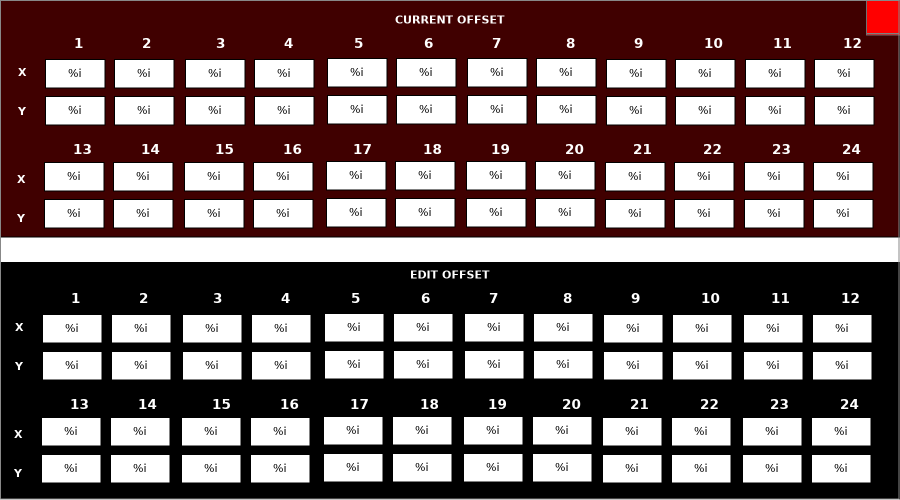
VISUALIZATION MOffset_1  // 900x500
    RoundedRectangle (0,0 900x237)
    Label (0,0 900x40), "CURRENT OFFSET"
    Label (15,55 25x35), "X"
    RoundedRectangle (45,59 60x29), "%i", text variable: Status_GVL.RecipeLine[1].OffsetPattern.Offset_X[1]
    Label (71,26 25x35), "1"
    RoundedRectangle (114,59 60x29), "%i", text variable: Status_GVL.RecipeLine[1].OffsetPattern.Offset_X[2]
    Label (139,26 25x35), "2"
    RoundedRectangle (185,59 60x29), "%i", text variable: Status_GVL.RecipeLine[1].OffsetPattern.Offset_X[3]
    RoundedRectangle (254,59 60x29), "%i", text variable: Status_GVL.RecipeLine[1].OffsetPattern.Offset_X[4]
    Label (15,94 25x35), "Y"
    RoundedRectangle (327,58 60x29), "%i", text variable: Status_GVL.RecipeLine[1].OffsetPattern.Offset_X[5]
    RoundedRectangle (396,58 60x29), "%i", text variable: Status_GVL.RecipeLine[1].OffsetPattern.Offset_X[6]
    RoundedRectangle (467,58 60x29), "%i", text variable: Status_GVL.RecipeLine[1].OffsetPattern.Offset_X[7]
    RoundedRectangle (536,58 60x29), "%i", text variable: Status_GVL.RecipeLine[1].OffsetPattern.Offset_X[8]
    RoundedRectangle (606,59 60x29), "%i", text variable: Status_GVL.RecipeLine[1].OffsetPattern.Offset_X[9]
    RoundedRectangle (675,59 60x29), "%i", text variable: Status_GVL.RecipeLine[1].OffsetPattern.Offset_X[10]
    Label (213,26 25x35), "3"
    Label (281,26 25x35), "4"
    Label (351,26 25x35), "5"
    Label (421,26 25x35), "6"
    Label (489,26 25x35), "7"
    Label (563,26 25x35), "8"
    Label (631,26 25x35), "9"
    Label (701,26 25x35), "10"
    RoundedRectangle (45,96 60x29), "%i", text variable: Status_GVL.RecipeLine[1].OffsetPattern.Offset_Y[1]
    RoundedRectangle (114,96 60x29), "%i", text variable: Status_GVL.RecipeLine[1].OffsetPattern.Offset_Y[2]
    RoundedRectangle (185,96 60x29), "%i", text variable: Status_GVL.RecipeLine[1].OffsetPattern.Offset_Y[3]
    RoundedRectangle (254,96 60x29), "%i", text variable: Status_GVL.RecipeLine[1].OffsetPattern.Offset_Y[4]
    RoundedRectangle (327,95 60x29), "%i", text variable: Status_GVL.RecipeLine[1].OffsetPattern.Offset_Y[5]
    RoundedRectangle (396,95 60x29), "%i", text variable: Status_GVL.RecipeLine[1].OffsetPattern.Offset_Y[6]
    RoundedRectangle (467,95 60x29), "%i", text variable: Status_GVL.RecipeLine[1].OffsetPattern.Offset_Y[7]
    RoundedRectangle (536,95 60x29), "%i", text variable: Status_GVL.RecipeLine[1].OffsetPattern.Offset_Y[8]
    RoundedRectangle (606,96 60x29), "%i", text variable: Status_GVL.RecipeLine[1].OffsetPattern.Offset_Y[9]
    RoundedRectangle (675,96 60x29), "%i", text variable: Status_GVL.RecipeLine[1].OffsetPattern.Offset_Y[10]
    Label (14,162 25x35), "X"
    RoundedRectangle (44,162 60x29), "%i", text variable: Status_GVL.RecipeLine[1].OffsetPattern.Offset_X[13]
    RoundedRectangle (113,162 60x29), "%i", text variable: Status_GVL.RecipeLine[1].OffsetPattern.Offset_X[14]
    RoundedRectangle (184,162 60x29), "%i", text variable: Status_GVL.RecipeLine[1].OffsetPattern.Offset_X[15]
    RoundedRectangle (253,162 60x29), "%i", text variable: Status_GVL.RecipeLine[1].OffsetPattern.Offset_X[16]
    Label (14,201 25x35), "Y"
    RoundedRectangle (326,161 60x29), "%i", text variable: Status_GVL.RecipeLine[1].OffsetPattern.Offset_X[17]
    RoundedRectangle (395,161 60x29), "%i", text variable: Status_GVL.RecipeLine[1].OffsetPattern.Offset_X[18]
    RoundedRectangle (466,161 60x29), "%i", text variable: Status_GVL.RecipeLine[1].OffsetPattern.Offset_X[19]
    RoundedRectangle (535,161 60x29), "%i", text variable: Status_GVL.RecipeLine[1].OffsetPattern.Offset_X[20]
    RoundedRectangle (605,162 60x29), "%i", text variable: Status_GVL.RecipeLine[1].OffsetPattern.Offset_X[21]
    RoundedRectangle (674,162 60x29), "%i", text variable: Status_GVL.RecipeLine[1].OffsetPattern.Offset_X[22]
    RoundedRectangle (44,199 60x29), "%i", text variable: Status_GVL.RecipeLine[1].OffsetPattern.Offset_Y[13]
    RoundedRectangle (113,199 60x29), "%i", text variable: Status_GVL.RecipeLine[1].OffsetPattern.Offset_Y[14]
    RoundedRectangle (184,199 60x29), "%i", text variable: Status_GVL.RecipeLine[1].OffsetPattern.Offset_Y[15]
    RoundedRectangle (253,199 60x29), "%i", text variable: Status_GVL.RecipeLine[1].OffsetPattern.Offset_Y[16]
    RoundedRectangle (326,198 60x29), "%i", text variable: Status_GVL.RecipeLine[1].OffsetPattern.Offset_Y[17]
    RoundedRectangle (395,198 60x29), "%i", text variable: Status_GVL.RecipeLine[1].OffsetPattern.Offset_Y[18]
    RoundedRectangle (466,198 60x29), "%i", text variable: Status_GVL.RecipeLine[1].OffsetPattern.Offset_Y[19]
    RoundedRectangle (535,198 60x29), "%i", text variable: Status_GVL.RecipeLine[1].OffsetPattern.Offset_Y[20]
    RoundedRectangle (605,199 60x29), "%i", text variable: Status_GVL.RecipeLine[1].OffsetPattern.Offset_Y[21]
    RoundedRectangle (674,199 60x29), "%i", text variable: Status_GVL.RecipeLine[1].OffsetPattern.Offset_Y[22]
    Label (70,132 25x35), "13"
    Label (138,132 25x35), "14"
    Label (212,132 25x35), "15"
    Label (280,132 25x35), "16"
    Label (350,132 25x35), "17"
    Label (420,132 25x35), "18"
    Label (488,132 25x35), "19"
    Label (562,132 25x35), "20"
    Label (630,132 25x35), "21"
    Label (700,132 25x35), "22"
    RoundedRectangle (0,262 900x237)
    Label (0,255 900x40), "EDIT OFFSET"
    Label (12,310 25x35), "X"
    RoundedRectangle (42,314 60x29), "%i", text variable: HMI_GVL.arRecipeHMI[1].OffsetPattern.Offset_X[1], input disabled if: Status_GVL.StsEdit[1]
        OnMouseClick: write the text variable via Default
    Label (68,281 25x35), "1"
    RoundedRectangle (111,314 60x29), "%i", text variable: HMI_GVL.arRecipeHMI[1].OffsetPattern.Offset_X[2], input disabled if: Status_GVL.StsEdit[1]
        OnMouseClick: write the text variable via Default
    Label (136,281 25x35), "2"
    RoundedRectangle (182,314 60x29), "%i", text variable: HMI_GVL.arRecipeHMI[1].OffsetPattern.Offset_X[3], input disabled if: Status_GVL.StsEdit[1]
        OnMouseClick: write the text variable via Default
    RoundedRectangle (251,314 60x29), "%i", text variable: HMI_GVL.arRecipeHMI[1].OffsetPattern.Offset_X[4], input disabled if: Status_GVL.StsEdit[1]
        OnMouseClick: write the text variable via Default
    Label (12,349 25x35), "Y"
    RoundedRectangle (324,313 60x29), "%i", text variable: HMI_GVL.arRecipeHMI[1].OffsetPattern.Offset_X[5], input disabled if: Status_GVL.StsEdit[1]
        OnMouseClick: write the text variable via Default
    RoundedRectangle (393,313 60x29), "%i", text variable: HMI_GVL.arRecipeHMI[1].OffsetPattern.Offset_X[6], input disabled if: Status_GVL.StsEdit[1]
        OnMouseClick: write the text variable via Default
    RoundedRectangle (464,313 60x29), "%i", text variable: HMI_GVL.arRecipeHMI[1].OffsetPattern.Offset_X[7], input disabled if: Status_GVL.StsEdit[1]
        OnMouseClick: write the text variable via Default
    RoundedRectangle (533,313 60x29), "%i", text variable: HMI_GVL.arRecipeHMI[1].OffsetPattern.Offset_X[8], input disabled if: Status_GVL.StsEdit[1]
        OnMouseClick: write the text variable via Default
    RoundedRectangle (603,314 60x29), "%i", text variable: HMI_GVL.arRecipeHMI[1].OffsetPattern.Offset_X[9], input disabled if: Status_GVL.StsEdit[1]
        OnMouseClick: write the text variable via Default
    RoundedRectangle (672,314 60x29), "%i", text variable: HMI_GVL.arRecipeHMI[1].OffsetPattern.Offset_X[10], input disabled if: Status_GVL.StsEdit[1]
        OnMouseClick: write the text variable via Default
    Label (210,281 25x35), "3"
    Label (278,281 25x35), "4"
    Label (348,281 25x35), "5"
    Label (418,281 25x35), "6"
    Label (486,281 25x35), "7"
    Label (560,281 25x35), "8"
    Label (628,281 25x35), "9"
    Label (698,281 25x35), "10"
    RoundedRectangle (42,351 60x29), "%i", text variable: HMI_GVL.arRecipeHMI[1].OffsetPattern.Offset_Y[1], input disabled if: Status_GVL.StsEdit[1]
        OnMouseClick: write the text variable via Default
    RoundedRectangle (111,351 60x29), "%i", text variable: HMI_GVL.arRecipeHMI[1].OffsetPattern.Offset_Y[2], input disabled if: Status_GVL.StsEdit[1]
        OnMouseClick: write the text variable via Default
    RoundedRectangle (182,351 60x29), "%i", text variable: HMI_GVL.arRecipeHMI[1].OffsetPattern.Offset_Y[3], input disabled if: Status_GVL.StsEdit[1]
        OnMouseClick: write the text variable via Default
    RoundedRectangle (251,351 60x29), "%i", text variable: HMI_GVL.arRecipeHMI[1].OffsetPattern.Offset_Y[4], input disabled if: Status_GVL.StsEdit[1]
        OnMouseClick: write the text variable via Default
    RoundedRectangle (324,350 60x29), "%i", text variable: HMI_GVL.arRecipeHMI[1].OffsetPattern.Offset_Y[5], input disabled if: Status_GVL.StsEdit[1]
        OnMouseClick: write the text variable via Default
    RoundedRectangle (393,350 60x29), "%i", text variable: HMI_GVL.arRecipeHMI[1].OffsetPattern.Offset_Y[6], input disabled if: Status_GVL.StsEdit[1]
        OnMouseClick: write the text variable via Default
    RoundedRectangle (464,350 60x29), "%i", text variable: HMI_GVL.arRecipeHMI[1].OffsetPattern.Offset_Y[7], input disabled if: Status_GVL.StsEdit[1]
        OnMouseClick: write the text variable via Default
    RoundedRectangle (533,350 60x29), "%i", text variable: HMI_GVL.arRecipeHMI[1].OffsetPattern.Offset_Y[8], input disabled if: Status_GVL.StsEdit[1]
        OnMouseClick: write the text variable via Default
    RoundedRectangle (603,351 60x29), "%i", text variable: HMI_GVL.arRecipeHMI[1].OffsetPattern.Offset_Y[9], input disabled if: Status_GVL.StsEdit[1]
        OnMouseClick: write the text variable via Default
    RoundedRectangle (672,351 60x29), "%i", text variable: HMI_GVL.arRecipeHMI[1].OffsetPattern.Offset_Y[10], input disabled if: Status_GVL.StsEdit[1]
        OnMouseClick: write the text variable via Default
    Label (11,417 25x35), "X"
    RoundedRectangle (41,417 60x29), "%i", text variable: HMI_GVL.arRecipeHMI[1].OffsetPattern.Offset_X[13], input disabled if: Status_GVL.StsEdit[1]
        OnMouseClick: write the text variable via Default
    RoundedRectangle (110,417 60x29), "%i", text variable: HMI_GVL.arRecipeHMI[1].OffsetPattern.Offset_X[14], input disabled if: Status_GVL.StsEdit[1]
        OnMouseClick: write the text variable via Default
    RoundedRectangle (181,417 60x29), "%i", text variable: HMI_GVL.arRecipeHMI[1].OffsetPattern.Offset_X[15], input disabled if: Status_GVL.StsEdit[1]
        OnMouseClick: write the text variable via Default
    RoundedRectangle (250,417 60x29), "%i", text variable: HMI_GVL.arRecipeHMI[1].OffsetPattern.Offset_X[16], input disabled if: Status_GVL.StsEdit[1]
        OnMouseClick: write the text variable via Default
    Label (11,456 25x35), "Y"
    RoundedRectangle (323,416 60x29), "%i", text variable: HMI_GVL.arRecipeHMI[1].OffsetPattern.Offset_X[17], input disabled if: Status_GVL.StsEdit[1]
        OnMouseClick: write the text variable via Default
    RoundedRectangle (392,416 60x29), "%i", text variable: HMI_GVL.arRecipeHMI[1].OffsetPattern.Offset_X[18], input disabled if: Status_GVL.StsEdit[1]
        OnMouseClick: write the text variable via Default
    RoundedRectangle (463,416 60x29), "%i", text variable: HMI_GVL.arRecipeHMI[1].OffsetPattern.Offset_X[19], input disabled if: Status_GVL.StsEdit[1]
        OnMouseClick: write the text variable via Default
    RoundedRectangle (532,416 60x29), "%i", text variable: HMI_GVL.arRecipeHMI[1].OffsetPattern.Offset_X[20], input disabled if: Status_GVL.StsEdit[1]
        OnMouseClick: write the text variable via Default
    RoundedRectangle (602,417 60x29), "%i", text variable: HMI_GVL.arRecipeHMI[1].OffsetPattern.Offset_X[21], input disabled if: Status_GVL.StsEdit[1]
        OnMouseClick: write the text variable via Default
    RoundedRectangle (671,417 60x29), "%i", text variable: HMI_GVL.arRecipeHMI[1].OffsetPattern.Offset_X[22], input disabled if: Status_GVL.StsEdit[1]
        OnMouseClick: write the text variable via Default
    RoundedRectangle (41,454 60x29), "%i", text variable: HMI_GVL.arRecipeHMI[1].OffsetPattern.Offset_Y[13], input disabled if: Status_GVL.StsEdit[1]
        OnMouseClick: write the text variable via Default
    RoundedRectangle (110,454 60x29), "%i", text variable: HMI_GVL.arRecipeHMI[1].OffsetPattern.Offset_Y[14], input disabled if: Status_GVL.StsEdit[1]
        OnMouseClick: write the text variable via Default
    RoundedRectangle (181,454 60x29), "%i", text variable: HMI_GVL.arRecipeHMI[1].OffsetPattern.Offset_Y[15], input disabled if: Status_GVL.StsEdit[1]
        OnMouseClick: write the text variable via Default
    RoundedRectangle (250,454 60x29), "%i", text variable: HMI_GVL.arRecipeHMI[1].OffsetPattern.Offset_Y[16], input disabled if: Status_GVL.StsEdit[1]
        OnMouseClick: write the text variable via Default
    RoundedRectangle (323,453 60x29), "%i", text variable: HMI_GVL.arRecipeHMI[1].OffsetPattern.Offset_Y[17], input disabled if: Status_GVL.StsEdit[1]
        OnMouseClick: write the text variable via Default
    RoundedRectangle (392,453 60x29), "%i", text variable: HMI_GVL.arRecipeHMI[1].OffsetPattern.Offset_Y[18], input disabled if: Status_GVL.StsEdit[1]
        OnMouseClick: write the text variable via Default
    RoundedRectangle (463,453 60x29), "%i", text variable: HMI_GVL.arRecipeHMI[1].OffsetPattern.Offset_Y[19], input disabled if: Status_GVL.StsEdit[1]
        OnMouseClick: write the text variable via Default
    RoundedRectangle (532,453 60x29), "%i", text variable: HMI_GVL.arRecipeHMI[1].OffsetPattern.Offset_Y[20], input disabled if: Status_GVL.StsEdit[1]
        OnMouseClick: write the text variable via Default
    RoundedRectangle (602,454 60x29), "%i", text variable: HMI_GVL.arRecipeHMI[1].OffsetPattern.Offset_Y[21], input disabled if: Status_GVL.StsEdit[1]
        OnMouseClick: write the text variable via Default
    RoundedRectangle (671,454 60x29), "%i", text variable: HMI_GVL.arRecipeHMI[1].OffsetPattern.Offset_Y[22], input disabled if: Status_GVL.StsEdit[1]
        OnMouseClick: write the text variable via Default
    Label (67,387 25x35), "13"
    Label (135,387 25x35), "14"
    Label (209,387 25x35), "15"
    Label (277,387 25x35), "16"
    Label (347,387 25x35), "17"
    Label (417,387 25x35), "18"
    Label (485,387 25x35), "19"
    Label (559,387 25x35), "20"
    Label (627,387 25x35), "21"
    Label (697,387 25x35), "22"
    Button (866,0 35x35), image: VisuSymbols.Symbols.Wrong
        OnMouseClick: CloseDialog Dialog=MOffset_1, Result=OK, NumpadKeypadSet=True
    RoundedRectangle (745,59 60x29), "%i", text variable: Status_GVL.RecipeLine[1].OffsetPattern.Offset_X[11]
    RoundedRectangle (814,59 60x29), "%i", text variable: Status_GVL.RecipeLine[1].OffsetPattern.Offset_X[12]
    Label (770,26 25x35), "11"
    Label (840,26 25x35), "12"
    RoundedRectangle (745,96 60x29), "%i", text variable: Status_GVL.RecipeLine[1].OffsetPattern.Offset_Y[11]
    RoundedRectangle (814,96 60x29), "%i", text variable: Status_GVL.RecipeLine[1].OffsetPattern.Offset_Y[12]
    RoundedRectangle (744,162 60x29), "%i", text variable: Status_GVL.RecipeLine[1].OffsetPattern.Offset_X[23]
    RoundedRectangle (813,162 60x29), "%i", text variable: Status_GVL.RecipeLine[1].OffsetPattern.Offset_X[24]
    RoundedRectangle (744,199 60x29), "%i", text variable: Status_GVL.RecipeLine[1].OffsetPattern.Offset_Y[23]
    RoundedRectangle (813,199 60x29), "%i", text variable: Status_GVL.RecipeLine[1].OffsetPattern.Offset_Y[24]
    Label (769,132 25x35), "23"
    Label (839,132 25x35), "24"
    RoundedRectangle (743,314 60x29), "%i", text variable: HMI_GVL.arRecipeHMI[1].OffsetPattern.Offset_X[11], input disabled if: Status_GVL.StsEdit[1]
        OnMouseClick: write the text variable via Default
    RoundedRectangle (812,314 60x29), "%i", text variable: HMI_GVL.arRecipeHMI[1].OffsetPattern.Offset_X[12], input disabled if: Status_GVL.StsEdit[1]
        OnMouseClick: write the text variable via Default
    Label (768,281 25x35), "11"
    Label (838,281 25x35), "12"
    RoundedRectangle (743,351 60x29), "%i", text variable: HMI_GVL.arRecipeHMI[1].OffsetPattern.Offset_Y[11], input disabled if: Status_GVL.StsEdit[1]
        OnMouseClick: write the text variable via Default
    RoundedRectangle (812,351 60x29), "%i", text variable: HMI_GVL.arRecipeHMI[1].OffsetPattern.Offset_Y[12], input disabled if: Status_GVL.StsEdit[1]
        OnMouseClick: write the text variable via Default
    RoundedRectangle (742,417 60x29), "%i", text variable: HMI_GVL.arRecipeHMI[1].OffsetPattern.Offset_X[23], input disabled if: Status_GVL.StsEdit[1]
        OnMouseClick: write the text variable via Default
    RoundedRectangle (811,417 60x29), "%i", text variable: HMI_GVL.arRecipeHMI[1].OffsetPattern.Offset_X[24], input disabled if: Status_GVL.StsEdit[1]
        OnMouseClick: write the text variable via Default
    RoundedRectangle (742,454 60x29), "%i", text variable: HMI_GVL.arRecipeHMI[1].OffsetPattern.Offset_Y[23], input disabled if: Status_GVL.StsEdit[1]
        OnMouseClick: write the text variable via Default
    RoundedRectangle (811,454 60x29), "%i", text variable: HMI_GVL.arRecipeHMI[1].OffsetPattern.Offset_Y[24], input disabled if: Status_GVL.StsEdit[1]
        OnMouseClick: write the text variable via Default
    Label (767,387 25x35), "23"
    Label (837,387 25x35), "24"
END_VISUALIZATION

(* stored: Version 1.1.0.1, ProductVersion 3.1.4024.12
   Visu MOffset_1: Id {280c222d-123e-4465-aba4-00e176774835} *)
